// TIA Portal V19 export
DATA_BLOCK "CallEquipment_DB"   // DB136
AUTHOR : Siemens_FA_SUP
// stored: AssignedProDiagFB Unit2.EM1.ProDiag, InstanceOfName Unit2.Em6.CallEquipment, InstanceOfType FB, Namespace Unit2.Em6
"Unit2.Em6.CallEquipment"
   // VAR_IN_OUT
   //    unitStatus : "LAF_typeUnitStatus";
   //    unitAlarmDB : "LAF_typeAlarms";
   //    emFeedback : "LUC_typeEmFeedback";
   // END_VAR
   // VAR
   //    statUnitStatus { ExternalWritable := 'False'} : "LAF_typeUnitStatus";
   //    instJobExecute { ExternalWritable := 'False'} : "LAF_SelectJob";
   //    instJobStopping { ExternalWritable := 'False'; S7_SetPoint := 'True'} : "LAF_SelectJob";
   //    instJobStarting { ExternalWritable := 'False'; S7_SetPoint := 'True'} : "LAF_SelectJob";
   //    instJobHolding { ExternalWritable := 'False'; S7_SetPoint := 'True'} : "LAF_SelectJob";
   //    instJobUnHolding { ExternalWritable := 'False'; S7_SetPoint := 'True'} : "LAF_SelectJob";
   //    instJobReseting { ExternalWritable := 'False'; S7_SetPoint := 'True'} : "LAF_SelectJob";
   //    instSequence { ExternalWritable := 'False'} : "Unit2.Em6.Sequence";
   //    instManageBitAlarms { ExternalWritable := 'False'} : "LAF_ManageBitAlarms";
   //    instCm1Vfd207 { ExternalWritable := 'False'} : "LEXCHANGETRAY_RollerVfd";
   //    instCm2SignalTM { ExternalWritable := 'False'} : "LEXCHANGETRAY_U2Em6SingleTM";
   //    statLstUnitMode { ExternalWritable := 'False'; S7_SetPoint := 'True'} : DInt;
   // END_VAR
BEGIN
END_DATA_BLOCK
